TYPE ST_HMI_Historize :
STRUCT
	PSB				: ST_HMI_PowerMeas;
	Input			: ST_HMI_PowerMeas;
	Output			: ST_HMI_PowerMeas;
	Inverter		: ST_HMI_PowerMeas;
	Battery			: ST_HMI_PowerMeasDC;
	Charger			: ST_HMI_PowerMeas;
	DcCoupling		: ST_HMI_PowerMeasDC;
END_STRUCT
END_TYPE

(* stored: Version 1.1.0.1, ProductVersion 3.1.4026.18
   DUT ST_HMI_Historize: Id {51de7ebf-3a4c-4cc3-ba28-e052945c3e46} *)
